Staubli VAL3: killBlink.pgx

public program killBlink(string x_sDioName)
begin


  //destroy the task that is making the dio blinking...
  taskKill("blink_"+x_sDioName)
  wait(taskStatus("blink_"+x_sDioName)==-1)


end
